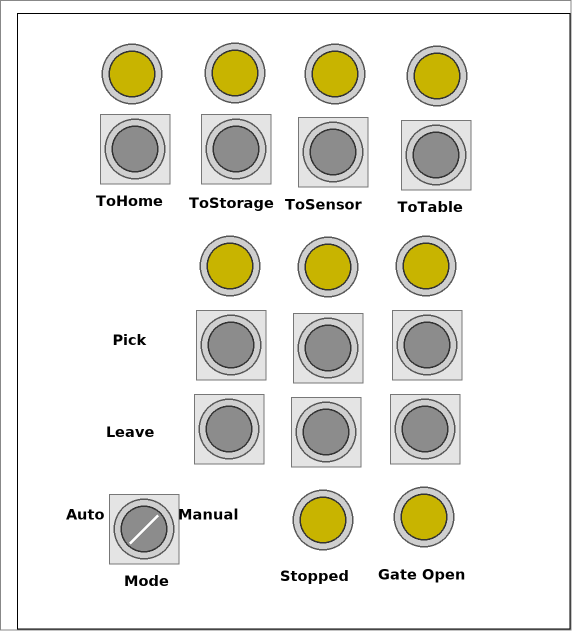
VISUALIZATION STNX00HMI  // 572x631
    RoundedRectangle (17,13 553x616)
    Label (62,498 47x33), "Auto"
    RotarySwitch (109,494 70x70), behaviour: TOGGLE, style: Switch-RotarySwitch-Gray
    Label (120,566 53x30), "Mode"
    Label (172,499 73x31), "Manual"
    PushSwitch (100,114 70x70), behaviour: TOGGLE, style: Switch-PushSwitch-Gray
    PushSwitch (201,114 70x70), behaviour: TOGGLE, style: Switch-PushSwitch-Gray
    PushSwitch (298,117 70x70), behaviour: TOGGLE, style: Switch-PushSwitch-Gray
    Label (87,184 85x34), "ToHome"
    Label (189,186 85x34), "ToStorage"
    Label (275,186 97x37), "ToSensor"
    PushSwitch (196,310 70x70), behaviour: TOGGLE, style: Switch-PushSwitch-Gray
    PushSwitch (293,313 70x70), behaviour: TOGGLE, style: Switch-PushSwitch-Gray
    Label (87,323 85x34), "Pick"
    PushSwitch (401,120 70x70), behaviour: TOGGLE, style: Switch-PushSwitch-Gray
    Label (388,190 85x34), "ToTable"
    Lamp1 (97,39 70x70), style: Lamp-Lamp1-Yellow
    Lamp1 (200,38 70x70), style: Lamp-Lamp1-Yellow
    Lamp1 (300,39 70x70), style: Lamp-Lamp1-Yellow
    Lamp1 (402,41 70x70), style: Lamp-Lamp1-Yellow
    Lamp1 (195,231 70x70), style: Lamp-Lamp1-Yellow
    Lamp1 (293,232 70x70), style: Lamp-Lamp1-Yellow
    Lamp1 (391,231 70x70), style: Lamp-Lamp1-Yellow
    PushSwitch (392,310 70x70), behaviour: TOGGLE, style: Switch-PushSwitch-Gray
    PushSwitch (194,394 70x70), behaviour: TOGGLE, style: Switch-PushSwitch-Gray
    PushSwitch (291,397 70x70), behaviour: TOGGLE, style: Switch-PushSwitch-Gray
    PushSwitch (390,394 70x70), behaviour: TOGGLE, style: Switch-PushSwitch-Gray
    Label (88,415 85x34), "Leave"
    Lamp1 (288,485 70x70), style: Lamp-Lamp1-Yellow
    Lamp1 (389,482 70x70), style: Lamp-Lamp1-Yellow
    Label (373,553 98x43), "Gate Open"
    Label (267,559 95x34), "Stopped"
END_VISUALIZATION

(* stored: Version 1.1.0.1, ProductVersion 3.1.4024.2
   Visu STNX00HMI: Id {a029b0e6-70c2-4e2e-a1cf-7e9ed73d1bdf} *)
